// TIA Portal V19 export
DATA_BLOCK "FC_Modbus_Arduino_DB"   // DB4
// stored: InstanceOfName FC_Modbus_Arduino, InstanceOfType FB
"FC_Modbus_Arduino"
   // VAR_INPUT
   //    Start_Feeder : Bool;
   // END_VAR
   // VAR_OUTPUT
   //    Feeder_Ready : Bool;
   // END_VAR
BEGIN
END_DATA_BLOCK
